// TIA Portal project "Sistema_semaforico2" (V15.1)

(* hardware
DEVICE "S7-1200 station_1"  S7-1200 Station
   slot 0: "Telaio di montaggio_0"  S7-1200 Rack  Rack  V1.0
   slot 1: "PLC_1"  CPU 1214C DC/DC/DC  6ES7 214-1AG40-0XB0  V4.2
*)

// ===== PLC "PLC_1"  CPU 1214C DC/DC/DC =====

VAR_GLOBAL   // PLC tag table "Tabella delle variabili standard"
   "P" AT %I0.0 : Bool;
   "verde1" AT %Q0.0 : Bool;
   "giallo1" AT %Q0.1 : Bool;
   "rosso1" AT %Q0.2 : Bool;
   "verde2" AT %Q0.3 : Bool;
   "giallo2" AT %Q0.4 : Bool;
   "rosso2" AT %Q0.5 : Bool;
END_VAR

VAR_GLOBAL CONSTANT   // PLC tag table "Tabella delle variabili standard"
   "tempoVerde" : Time := T#55s;
   "tempoRosso" : Time := T#60s;
   "TempoGiallo" : Time := T#5s;
END_VAR

DATA_BLOCK "variabili_stato"   // DB1
{ S7_Optimized_Access := 'TRUE' }
VERSION : 0.1
   VAR RETAIN
      home : Bool := true;
      VR : Bool;
      GR : Bool;
      RV : Bool;
      RG : Bool;
      RR : Bool;
      prenotato : Bool;
   END_VAR
BEGIN
END_DATA_BLOCK

// folder: System blocks/Program resources

DATA_BLOCK "IEC_Timer_0_DB"   // DB2
{ S7_Optimized_Access := 'TRUE' }
AUTHOR : Simatic
FAMILY : IEC
NAME : IEC_TMR
VERSION : 1.0
// stored: InstanceOfName IEC_TIMER
"IEC_TIMER"
BEGIN
END_DATA_BLOCK

DATA_BLOCK "IEC_Timer_0_DB_1"   // DB3
{ S7_Optimized_Access := 'TRUE' }
AUTHOR : Simatic
FAMILY : IEC
NAME : IEC_TMR
VERSION : 1.0
// stored: InstanceOfName IEC_TIMER
"IEC_TIMER"
BEGIN
END_DATA_BLOCK

DATA_BLOCK "IEC_Timer_0_DB_2"   // DB4
{ S7_Optimized_Access := 'TRUE' }
AUTHOR : Simatic
FAMILY : IEC
NAME : IEC_TMR
VERSION : 1.0
// stored: InstanceOfName IEC_TIMER
"IEC_TIMER"
BEGIN
END_DATA_BLOCK

DATA_BLOCK "IEC_Timer_0_DB_3"   // DB5
{ S7_Optimized_Access := 'TRUE' }
AUTHOR : Simatic
FAMILY : IEC
NAME : IEC_TMR
VERSION : 1.0
// stored: InstanceOfName IEC_TIMER
"IEC_TIMER"
BEGIN
END_DATA_BLOCK

DATA_BLOCK "IEC_Timer_0_DB_4"   // DB6
{ S7_Optimized_Access := 'TRUE' }
AUTHOR : Simatic
FAMILY : IEC
NAME : IEC_TMR
VERSION : 1.0
// stored: InstanceOfName IEC_TIMER
"IEC_TIMER"
BEGIN
END_DATA_BLOCK

// folder: (top level)

ORGANIZATION_BLOCK "Main"   // OB1, LAD, ProgramCycle
TITLE = "Main Program Sweep (Cycle)"
{ S7_Optimized_Access := 'TRUE' }
VERSION : 0.1
   VAR_INPUT
      Initial_Call : Bool;   // Initial call of this OB
      Remanence : Bool;   // =True, if remanent data are available
   END_VAR
   VAR_TEMP   // added for the SCL form of the ladder/FBD networks
      _w1 : Bool;
   END_VAR
BEGIN

REGION Network 1
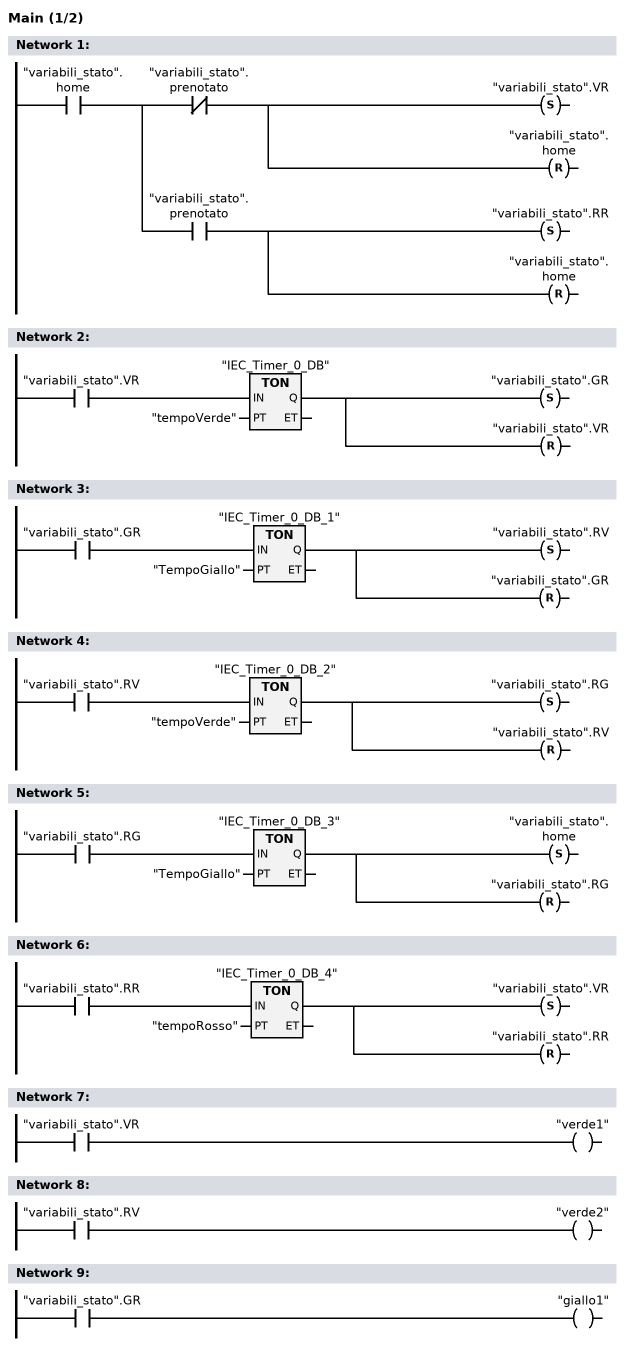
   RUNG wire#powerrail
      Contact( "variabili_stato".home )
      wire#w1
      I_Contact( "variabili_stato".prenotato )
      wire#w2
      S_Coil( "variabili_stato".VR )
   END_RUNG
   RUNG wire#w2
      R_Coil( "variabili_stato".home )
   END_RUNG
   RUNG wire#w1
      Contact( "variabili_stato".prenotato )
      wire#w3
      S_Coil( "variabili_stato".RR )
   END_RUNG
   RUNG wire#w3
      R_Coil( "variabili_stato".home )
   END_RUNG
   // the same network as SCL:
   IF "variabili_stato".home AND NOT "variabili_stato".prenotato THEN "variabili_stato".VR := TRUE; END_IF;
   #_w1 := "variabili_stato".home;
   IF "variabili_stato".home AND NOT "variabili_stato".prenotato THEN
       "variabili_stato".home := FALSE;
   END_IF;
   IF #_w1 AND "variabili_stato".prenotato THEN
       "variabili_stato".RR := TRUE;
       "variabili_stato".home := FALSE;
   END_IF;
END_REGION

REGION Network 2
   "IEC_Timer_0_DB".TON(IN := "variabili_stato".VR, PT := "tempoVerde");
   IF "IEC_Timer_0_DB".Q THEN
       "variabili_stato".GR := TRUE;
       "variabili_stato".VR := FALSE;
   END_IF;
END_REGION

REGION Network 3
   "IEC_Timer_0_DB_1".TON(IN := "variabili_stato".GR, PT := "TempoGiallo");
   IF "IEC_Timer_0_DB_1".Q THEN
       "variabili_stato".RV := TRUE;
       "variabili_stato".GR := FALSE;
   END_IF;
END_REGION

REGION Network 4
   "IEC_Timer_0_DB_2".TON(IN := "variabili_stato".RV, PT := "tempoVerde");
   IF "IEC_Timer_0_DB_2".Q THEN
       "variabili_stato".RG := TRUE;
       "variabili_stato".RV := FALSE;
   END_IF;
END_REGION

REGION Network 5
   "IEC_Timer_0_DB_3".TON(IN := "variabili_stato".RG, PT := "TempoGiallo");
   IF "IEC_Timer_0_DB_3".Q THEN
       "variabili_stato".home := TRUE;
       "variabili_stato".RG := FALSE;
   END_IF;
END_REGION

REGION Network 6
   "IEC_Timer_0_DB_4".TON(IN := "variabili_stato".RR, PT := "tempoRosso");
   IF "IEC_Timer_0_DB_4".Q THEN
       "variabili_stato".VR := TRUE;
       "variabili_stato".RR := FALSE;
   END_IF;
END_REGION

REGION Network 7
   RUNG wire#powerrail
      Contact( "variabili_stato".VR )
      Coil( "verde1" )
   END_RUNG
   // the same network as SCL:
   "verde1" := "variabili_stato".VR;
END_REGION

REGION Network 8
   RUNG wire#powerrail
      Contact( "variabili_stato".RV )
      Coil( "verde2" )
   END_RUNG
   // the same network as SCL:
   "verde2" := "variabili_stato".RV;
END_REGION

REGION Network 9
   RUNG wire#powerrail
      Contact( "variabili_stato".GR )
      Coil( "giallo1" )
   END_RUNG
   // the same network as SCL:
   "giallo1" := "variabili_stato".GR;
END_REGION

REGION Network 10
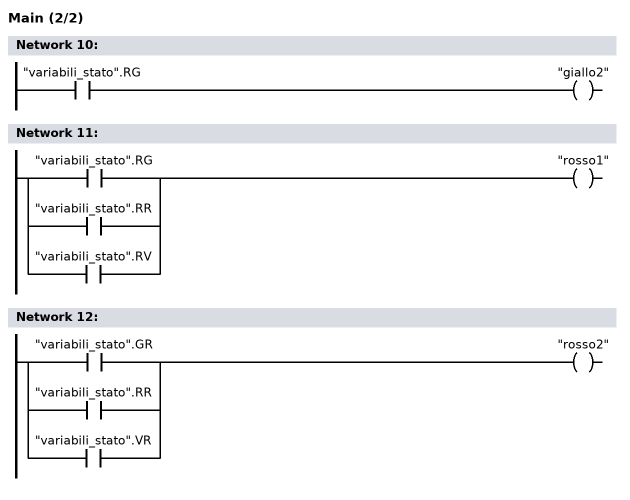
   RUNG wire#powerrail
      Contact( "variabili_stato".RG )
      Coil( "giallo2" )
   END_RUNG
   // the same network as SCL:
   "giallo2" := "variabili_stato".RG;
END_REGION

REGION Network 11
   RUNG wire#powerrail
      Contact( "variabili_stato".RG )
      wire#w1
      Coil( "rosso1" )
   END_RUNG
   RUNG wire#powerrail
      Contact( "variabili_stato".RR )
   END_RUNG wire#w1
   RUNG wire#powerrail
      Contact( "variabili_stato".RV )
   END_RUNG wire#w1
   // the same network as SCL:
   "rosso1" := "variabili_stato".RG OR "variabili_stato".RR OR "variabili_stato".RV;
END_REGION

REGION Network 12
   RUNG wire#powerrail
      Contact( "variabili_stato".GR )
      wire#w1
      Coil( "rosso2" )
   END_RUNG
   RUNG wire#powerrail
      Contact( "variabili_stato".RR )
   END_RUNG wire#w1
   RUNG wire#powerrail
      Contact( "variabili_stato".VR )
   END_RUNG wire#w1
   // the same network as SCL:
   "rosso2" := "variabili_stato".GR OR "variabili_stato".RR OR "variabili_stato".VR;
END_REGION
END_ORGANIZATION_BLOCK

ORGANIZATION_BLOCK "task_prenotato"   // OB40, LAD, HWProcessInterrupt
{ S7_Optimized_Access := 'TRUE' }
VERSION : 0.1
   VAR_INPUT
      LADDR : Hw_Io;   // Hardware identifier
      USI : Word;   // User structure identifier
      IChannel : USInt;   // Interrupt channel number
      EventType : Byte;   // EventType
   END_VAR
BEGIN

REGION Network 1
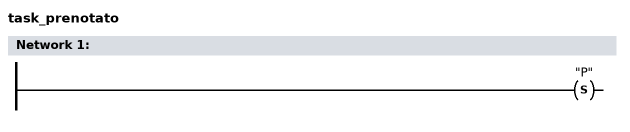
   RUNG wire#powerrail
      S_Coil( "P" )
   END_RUNG
   // the same network as SCL:
   "P" := TRUE;
END_REGION
END_ORGANIZATION_BLOCK